{attribute 'GeneratedUsingTerminal: EL3632-0000-0016'}
{attribute addProperty BoxType "EL3632-0000-0016"}
{attribute addProperty Id "STATUSAT %I*STATUS_B07533568"}
{attribute addProperty CRC "1971471493"}
{attribute addProperty Size "8"}
TYPE Ch2_Status_75824485 EXTENDS InputBase_8311D824 :
STRUCT
	{attribute addProperty Name "STATUS"}
	STATUS AT %I* : STATUS_B0753356;
END_STRUCT
END_TYPE

(* stored: Version 1.2.0.0, ProductVersion 3.1.4024.11
   DUT Ch2_Status_75824485: Id {1da6bd4d-cbe2-4887-9e8d-95159e1051ff} *)
